TYPE CalibrateConfig :
STRUCT
	CalibratePath : STRING;
	CalibrateHeaderNodeXml : STRING;
END_STRUCT
END_TYPE

(* stored: Version 1.1.0.1, ProductVersion 3.1.4024.3
   DUT CalibrateConfig: Id {0913e5b8-975c-406c-903d-1df1226c34f3} *)
